DATA_BLOCK "DB2039_TQ"
TITLE = DB2039_TQ
{ S7_Optimized_Access := 'FALSE' }
AUTHOR : HCR
FAMILY : ZeusControl
VERSION : 1.0
//Bloque de datos dispositivo TQ.
   STRUCT
      TQ { S7_SetPoint := 'False'} : Array[0.."N_MAX_DISP_TQ"] of "UDT_ZC_DISP_TQ";
      Mux { S7_SetPoint := 'False'} : Array[0.."N_MAX_MUX_DISP"] of "UDT_ZC_DISP_MUX_TQ";
      Agrup : Array[0.."N_MAX_DISP_AGRUP"] of "UDT_ZC_DISP_AGRUP";
   END_STRUCT;


BEGIN
   TQ[0].Hmi_Estado := 0;
   TQ[0].Estado_TanqueVacio := FALSE;
   TQ[0].Estado_PocisionAltura := FALSE;
   TQ[0].Estado_NivelBajo := FALSE;
   TQ[0].Estado_NivelAlto := FALSE;
   TQ[0].Estado_BocaHombre := FALSE;
   TQ[0].Estado_Mezcla := FALSE;
   TQ[0].Estado_ComOk := FALSE;
   TQ[0].Alarmas_NivelBajo := FALSE;
   TQ[0].Alarmas_NivelAlto := FALSE;
   TQ[0].Alarmas_BocaHombre := FALSE;
   TQ[0].Alarmas_Instrumentacion := FALSE;
   TQ[0].Alarmas_Parametros := FALSE;
   TQ[0].Alarmas_General := FALSE;
   TQ[0].Alarmas_Capacidad := FALSE;
   TQ[0].Orden_Temperatura := FALSE;
   TQ[0].Orden_Agitacion := FALSE;
   TQ[0].Orden_CIP := FALSE;
   TQ[0].Orden_Producto := FALSE;
   TQ[0].Orden_CambioEstado := FALSE;
   TQ[0].Orden_CambioProd1 := FALSE;
   TQ[0].Orden_CambioProd2 := FALSE;
   TQ[0].Config_Habilitar := FALSE;
   TQ[0].Config_HabilitarControlAgitacion := TRUE;
   TQ[0].Config_HabilitarControlTemp := TRUE;
   TQ[0].Config_HabilitarCamisa := TRUE;
   TQ[0].Config_HabilitarAgitador := TRUE;
   TQ[0].Config_HabilitarAlarmas := FALSE;
   TQ[0].Config_HabilitarCalculoVol := FALSE;
   TQ[0].Config_TipoControlTemperatura := FALSE;
   TQ[0].Aux_VisConsignaTemperatura := FALSE;
   TQ[0].Aux_PulsoAlternarAG := FALSE;
   TQ[0].Aux_MemOrdenAgitador := FALSE;
   TQ[0].Aux_MemOrdenTemperatura := FALSE;
   TQ[0].Aux_MemOrdenProducto := FALSE;
   TQ[0].Aux_MemEstadoCIP := FALSE;
   TQ[0].Aux_CipOK := FALSE;
   TQ[0].Orden_ParoControlAgitador := FALSE;
   TQ[0].Orden_ParoControlTemp := FALSE;
   TQ[0].R_Bool_6 := FALSE;
   TQ[0].R_Bool_8 := FALSE;
   TQ[0].Config_GrupoAlarma := 0;
   TQ[0].Estado_EA_Nivel := 0;
   TQ[0].Estado_EA_Temperatura := 0;
   TQ[0].Estado_Tanque := 0;
   TQ[0].Estado_TanqueNuevo := 0;
   TQ[0].Estado_Producto1 := 0;
   TQ[0].Estado_Producto2 := 0;
   TQ[0].Estado_ProductoNuevo := 0;
   TQ[0].Estado_Volumen := 0.0;
   TQ[0].Estado_Presion := 0.0;
   TQ[0].Estado_Altura := 0.0;
   TQ[0].Orden_TipoProducto := 0;
   TQ[0].Orden_ConsignaAgitador := 0.0;
   TQ[0].Config_NumeroEANivel := 0;
   TQ[0].Config_NumeroEATemp := 0;
   TQ[0].Config_NumeroLL := 0;
   TQ[0].Config_NumeroHL := 0;
   TQ[0].Config_NumeroBH := 0;
   TQ[0].Config_NumeroVA := 0;
   TQ[0].Config_NumeroAG := 0;
   TQ[0].Config_TipoAgitacionTiempo := 0;
   TQ[0].Config_TipoAgitacionVelocidad := 0;
   TQ[0].Config_TipoAgitador := 0;
   TQ[0].Config_EscaladoMinTarjeta := 0;
   TQ[0].Config_EscaladoMaxTarjeta := 27648;
   TQ[0].Config_EscaladoMinIngenieria := 0.0;
   TQ[0].Config_EscaladoMaxIngenieria := 0.1;
   TQ[0].Config_ConsignaTemperatura := 0.0;
   TQ[0].Config_HisteresisTemperatura := 0.0;
   TQ[0].Config_VolumenMinControlTemp := 0.0;
   TQ[0].Config_VolumenMaxControlTemp := 0.0;
   TQ[0].Config_VolumenMinControlAgitador := 0.0;
   TQ[0].Config_VolumenMaxControlAgitador := 0.0;
   TQ[0].Config_VolumenTanqueVacio := 0.0;
   TQ[0].Config_VelocidadMinAgitador := 0.0;
   TQ[0].Config_VelocidadMaxAgitador := 0.0;
   TQ[0].Config_VelocidadFijaAgitador := 0.0;
   TQ[0].Config_CapacidadTanque := 0.0;
   TQ[0].Config_DiametroCilindro := 0.0;
   TQ[0].Config_AlturaCilindro := 0.0;
   TQ[0].Config_DiametroConoInferior := 0.0;
   TQ[0].Config_AnguloCono := 0.0;
   TQ[0].Config_AlturaCono := 0.0;
   TQ[0].Tiempos_AgitadorONConsigna := 0;
   TQ[0].Tiempos_AgitadorONActual := 0;
   TQ[0].Tiempos_AgitadorOFFConsigna := 0;
   TQ[0].Tiempos_AgitadorOFFActual := 0;
   TQ[0].Tiempos_TiempoProducto.Hora := 0;
   TQ[0].Tiempos_TiempoProducto.Minuto := 0;
   TQ[0].Tiempos_TiempoProducto.Segundo := 0;
   TQ[0].Tiempos_TiempoLimpio.Hora := 0;
   TQ[0].Tiempos_TiempoLimpio.Minuto := 0;
   TQ[0].Tiempos_TiempoLimpio.Segundo := 0;
   TQ[0].Tiempos_RetTanqueVacio.SP := 5;
   TQ[0].Tiempos_RetTanqueVacio.ET := 0;
   TQ[0].Tiempos_RetTanqueVacio.IN := FALSE;
   TQ[0].Tiempos_RetTanqueVacio.Q := FALSE;
   TQ[0].Aux_ValorTarjetaNivel := 0;
   TQ[0].Aux_ValorIngeneriaTemperatura := 0.0;
   TQ[1].Hmi_Estado := 0;
   TQ[1].Estado_TanqueVacio := TRUE;
   TQ[1].Estado_PocisionAltura := FALSE;
   TQ[1].Estado_NivelBajo := FALSE;
   TQ[1].Estado_NivelAlto := FALSE;
   TQ[1].Estado_BocaHombre := TRUE;
   TQ[1].Estado_Mezcla := FALSE;
   TQ[1].Estado_ComOk := TRUE;
   TQ[1].Alarmas_NivelBajo := FALSE;
   TQ[1].Alarmas_NivelAlto := FALSE;
   TQ[1].Alarmas_BocaHombre := FALSE;
   TQ[1].Alarmas_Instrumentacion := FALSE;
   TQ[1].Alarmas_Parametros := FALSE;
   TQ[1].Alarmas_General := FALSE;
   TQ[1].Alarmas_Capacidad := FALSE;
   TQ[1].Orden_Temperatura := FALSE;
   TQ[1].Orden_Agitacion := FALSE;
   TQ[1].Orden_CIP := FALSE;
   TQ[1].Orden_Producto := FALSE;
   TQ[1].Orden_CambioEstado := FALSE;
   TQ[1].Orden_CambioProd1 := FALSE;
   TQ[1].Orden_CambioProd2 := FALSE;
   TQ[1].Config_Habilitar := TRUE;
   TQ[1].Config_HabilitarControlAgitacion := TRUE;
   TQ[1].Config_HabilitarControlTemp := TRUE;
   TQ[1].Config_HabilitarCamisa := TRUE;
   TQ[1].Config_HabilitarAgitador := TRUE;
   TQ[1].Config_HabilitarAlarmas := FALSE;
   TQ[1].Config_HabilitarCalculoVol := FALSE;
   TQ[1].Config_TipoControlTemperatura := TRUE;
   TQ[1].Aux_VisConsignaTemperatura := FALSE;
   TQ[1].Aux_PulsoAlternarAG := TRUE;
   TQ[1].Aux_MemOrdenAgitador := FALSE;
   TQ[1].Aux_MemOrdenTemperatura := FALSE;
   TQ[1].Aux_MemOrdenProducto := FALSE;
   TQ[1].Aux_MemEstadoCIP := FALSE;
   TQ[1].Aux_CipOK := FALSE;
   TQ[1].Orden_ParoControlAgitador := FALSE;
   TQ[1].Orden_ParoControlTemp := FALSE;
   TQ[1].R_Bool_6 := FALSE;
   TQ[1].R_Bool_8 := FALSE;
   TQ[1].Config_GrupoAlarma := 0;
   TQ[1].Estado_EA_Nivel := 1;
   TQ[1].Estado_EA_Temperatura := 1;
   TQ[1].Estado_Tanque := 2;
   TQ[1].Estado_TanqueNuevo := 1;
   TQ[1].Estado_Producto1 := 0;
   TQ[1].Estado_Producto2 := 0;
   TQ[1].Estado_ProductoNuevo := 1;
   TQ[1].Estado_Volumen := 0.0;
   TQ[1].Estado_Presion := 0.0;
   TQ[1].Estado_Altura := 0.0;
   TQ[1].Orden_TipoProducto := 1;
   TQ[1].Orden_ConsignaAgitador := 0.0;
   TQ[1].Config_NumeroEANivel := 9;
   TQ[1].Config_NumeroEATemp := 4;
   TQ[1].Config_NumeroLL := 0;
   TQ[1].Config_NumeroHL := 0;
   TQ[1].Config_NumeroBH := 8;
   TQ[1].Config_NumeroVA := 33;
   TQ[1].Config_NumeroAG := 4;
   TQ[1].Config_TipoAgitacionTiempo := 1;
   TQ[1].Config_TipoAgitacionVelocidad := 0;
   TQ[1].Config_TipoAgitador := 1;
   TQ[1].Config_EscaladoMinTarjeta := 0;
   TQ[1].Config_EscaladoMaxTarjeta := 27648;
   TQ[1].Config_EscaladoMinIngenieria := 0.0;
   TQ[1].Config_EscaladoMaxIngenieria := 0.1;
   TQ[1].Config_ConsignaTemperatura := 4.0;
   TQ[1].Config_HisteresisTemperatura := 1.0;
   TQ[1].Config_VolumenMinControlTemp := 200.0;
   TQ[1].Config_VolumenMaxControlTemp := 35000.0;
   TQ[1].Config_VolumenMinControlAgitador := 1600.0;
   TQ[1].Config_VolumenMaxControlAgitador := 30000.0;
   TQ[1].Config_VolumenTanqueVacio := 20.0;
   TQ[1].Config_VelocidadMinAgitador := 30.0;
   TQ[1].Config_VelocidadMaxAgitador := 85.0;
   TQ[1].Config_VelocidadFijaAgitador := 35.0;
   TQ[1].Config_CapacidadTanque := 30000.0;
   TQ[1].Config_DiametroCilindro := 0.0;
   TQ[1].Config_AlturaCilindro := 0.0;
   TQ[1].Config_DiametroConoInferior := 0.0;
   TQ[1].Config_AnguloCono := 0.0;
   TQ[1].Config_AlturaCono := 0.0;
   TQ[1].Tiempos_AgitadorONConsigna := 300;
   TQ[1].Tiempos_AgitadorONActual := 0;
   TQ[1].Tiempos_AgitadorOFFConsigna := 1200;
   TQ[1].Tiempos_AgitadorOFFActual := 0;
   TQ[1].Tiempos_TiempoProducto.Hora := 0;
   TQ[1].Tiempos_TiempoProducto.Minuto := 0;
   TQ[1].Tiempos_TiempoProducto.Segundo := 0;
   TQ[1].Tiempos_TiempoLimpio.Hora := 27;
   TQ[1].Tiempos_TiempoLimpio.Minuto := 30;
   TQ[1].Tiempos_TiempoLimpio.Segundo := 25;
   TQ[1].Tiempos_RetTanqueVacio.SP := 25;
   TQ[1].Tiempos_RetTanqueVacio.ET := 25;
   TQ[1].Tiempos_RetTanqueVacio.IN := TRUE;
   TQ[1].Tiempos_RetTanqueVacio.Q := TRUE;
   TQ[1].Aux_ValorTarjetaNivel := 0;
   TQ[1].Aux_ValorIngeneriaTemperatura := 26.19213;
   Mux[0].Habilitar := TRUE;
   Mux[0].ExisteCambio := FALSE;
   Mux[0].MaxVisible := FALSE;
   Mux[0].Index := 0;
   Mux[0].oldIndex := 0;
   Mux[0].TQ.Hmi_Estado := 0;
   Mux[0].TQ.Estado_TanqueVacio := FALSE;
   Mux[0].TQ.Estado_PocisionAltura := FALSE;
   Mux[0].TQ.Estado_NivelBajo := FALSE;
   Mux[0].TQ.Estado_NivelAlto := FALSE;
   Mux[0].TQ.Estado_BocaHombre := FALSE;
   Mux[0].TQ.Estado_Mezcla := FALSE;
   Mux[0].TQ.Estado_ComOk := FALSE;
   Mux[0].TQ.Alarmas_NivelBajo := FALSE;
   Mux[0].TQ.Alarmas_NivelAlto := FALSE;
   Mux[0].TQ.Alarmas_BocaHombre := FALSE;
   Mux[0].TQ.Alarmas_Instrumentacion := FALSE;
   Mux[0].TQ.Alarmas_Parametros := FALSE;
   Mux[0].TQ.Alarmas_General := FALSE;
   Mux[0].TQ.Alarmas_Capacidad := FALSE;
   Mux[0].TQ.Orden_Temperatura := FALSE;
   Mux[0].TQ.Orden_Agitacion := FALSE;
   Mux[0].TQ.Orden_CIP := FALSE;
   Mux[0].TQ.Orden_Producto := FALSE;
   Mux[0].TQ.Orden_CambioEstado := FALSE;
   Mux[0].TQ.Orden_CambioProd1 := FALSE;
   Mux[0].TQ.Orden_CambioProd2 := FALSE;
   Mux[0].TQ.Config_Habilitar := FALSE;
   Mux[0].TQ.Config_HabilitarControlAgitacion := TRUE;
   Mux[0].TQ.Config_HabilitarControlTemp := TRUE;
   Mux[0].TQ.Config_HabilitarCamisa := TRUE;
   Mux[0].TQ.Config_HabilitarAgitador := TRUE;
   Mux[0].TQ.Config_HabilitarAlarmas := FALSE;
   Mux[0].TQ.Config_HabilitarCalculoVol := FALSE;
   Mux[0].TQ.Config_TipoControlTemperatura := FALSE;
   Mux[0].TQ.Aux_VisConsignaTemperatura := FALSE;
   Mux[0].TQ.Aux_PulsoAlternarAG := FALSE;
   Mux[0].TQ.Aux_MemOrdenAgitador := FALSE;
   Mux[0].TQ.Aux_MemOrdenTemperatura := FALSE;
   Mux[0].TQ.Aux_MemOrdenProducto := FALSE;
   Mux[0].TQ.Aux_MemEstadoCIP := FALSE;
   Mux[0].TQ.Aux_CipOK := FALSE;
   Mux[0].TQ.Orden_ParoControlAgitador := FALSE;
   Mux[0].TQ.Orden_ParoControlTemp := FALSE;
   Mux[0].TQ.R_Bool_6 := FALSE;
   Mux[0].TQ.R_Bool_8 := FALSE;
   Mux[0].TQ.Config_GrupoAlarma := 0;
   Mux[0].TQ.Estado_EA_Nivel := 0;
   Mux[0].TQ.Estado_EA_Temperatura := 0;
   Mux[0].TQ.Estado_Tanque := 0;
   Mux[0].TQ.Estado_TanqueNuevo := 0;
   Mux[0].TQ.Estado_Producto1 := 0;
   Mux[0].TQ.Estado_Producto2 := 0;
   Mux[0].TQ.Estado_ProductoNuevo := 0;
   Mux[0].TQ.Estado_Volumen := 0.0;
   Mux[0].TQ.Estado_Presion := 0.0;
   Mux[0].TQ.Estado_Altura := 0.0;
   Mux[0].TQ.Orden_TipoProducto := 0;
   Mux[0].TQ.Orden_ConsignaAgitador := 0.0;
   Mux[0].TQ.Config_NumeroEANivel := 0;
   Mux[0].TQ.Config_NumeroEATemp := 0;
   Mux[0].TQ.Config_NumeroLL := 0;
   Mux[0].TQ.Config_NumeroHL := 0;
   Mux[0].TQ.Config_NumeroBH := 0;
   Mux[0].TQ.Config_NumeroVA := 0;
   Mux[0].TQ.Config_NumeroAG := 0;
   Mux[0].TQ.Config_TipoAgitacionTiempo := 0;
   Mux[0].TQ.Config_TipoAgitacionVelocidad := 0;
   Mux[0].TQ.Config_TipoAgitador := 0;
   Mux[0].TQ.Config_EscaladoMinTarjeta := 0;
   Mux[0].TQ.Config_EscaladoMaxTarjeta := 27648;
   Mux[0].TQ.Config_EscaladoMinIngenieria := 0.0;
   Mux[0].TQ.Config_EscaladoMaxIngenieria := 0.1;
   Mux[0].TQ.Config_ConsignaTemperatura := 0.0;
   Mux[0].TQ.Config_HisteresisTemperatura := 0.0;
   Mux[0].TQ.Config_VolumenMinControlTemp := 0.0;
   Mux[0].TQ.Config_VolumenMaxControlTemp := 0.0;
   Mux[0].TQ.Config_VolumenMinControlAgitador := 0.0;
   Mux[0].TQ.Config_VolumenMaxControlAgitador := 0.0;
   Mux[0].TQ.Config_VolumenTanqueVacio := 0.0;
   Mux[0].TQ.Config_VelocidadMinAgitador := 0.0;
   Mux[0].TQ.Config_VelocidadMaxAgitador := 0.0;
   Mux[0].TQ.Config_VelocidadFijaAgitador := 0.0;
   Mux[0].TQ.Config_CapacidadTanque := 0.0;
   Mux[0].TQ.Config_DiametroCilindro := 0.0;
   Mux[0].TQ.Config_AlturaCilindro := 0.0;
   Mux[0].TQ.Config_DiametroConoInferior := 0.0;
   Mux[0].TQ.Config_AnguloCono := 0.0;
   Mux[0].TQ.Config_AlturaCono := 0.0;
   Mux[0].TQ.Tiempos_AgitadorONConsigna := 0;
   Mux[0].TQ.Tiempos_AgitadorONActual := 0;
   Mux[0].TQ.Tiempos_AgitadorOFFConsigna := 0;
   Mux[0].TQ.Tiempos_AgitadorOFFActual := 0;
   Mux[0].TQ.Tiempos_TiempoProducto.Hora := 0;
   Mux[0].TQ.Tiempos_TiempoProducto.Minuto := 0;
   Mux[0].TQ.Tiempos_TiempoProducto.Segundo := 0;
   Mux[0].TQ.Tiempos_TiempoLimpio.Hora := 0;
   Mux[0].TQ.Tiempos_TiempoLimpio.Minuto := 0;
   Mux[0].TQ.Tiempos_TiempoLimpio.Segundo := 0;
   Mux[0].TQ.Tiempos_RetTanqueVacio.SP := 5;
   Mux[0].TQ.Tiempos_RetTanqueVacio.ET := 0;
   Mux[0].TQ.Tiempos_RetTanqueVacio.IN := FALSE;
   Mux[0].TQ.Tiempos_RetTanqueVacio.Q := FALSE;
   Mux[0].TQ.Aux_ValorTarjetaNivel := 0;
   Mux[0].TQ.Aux_ValorIngeneriaTemperatura := 0.0;
   Mux[1].Habilitar := TRUE;
   Mux[1].ExisteCambio := FALSE;
   Mux[1].MaxVisible := FALSE;
   Mux[1].Index := 0;
   Mux[1].oldIndex := 0;
   Mux[1].TQ.Hmi_Estado := 0;
   Mux[1].TQ.Estado_TanqueVacio := FALSE;
   Mux[1].TQ.Estado_PocisionAltura := FALSE;
   Mux[1].TQ.Estado_NivelBajo := FALSE;
   Mux[1].TQ.Estado_NivelAlto := FALSE;
   Mux[1].TQ.Estado_BocaHombre := FALSE;
   Mux[1].TQ.Estado_Mezcla := FALSE;
   Mux[1].TQ.Estado_ComOk := FALSE;
   Mux[1].TQ.Alarmas_NivelBajo := FALSE;
   Mux[1].TQ.Alarmas_NivelAlto := FALSE;
   Mux[1].TQ.Alarmas_BocaHombre := FALSE;
   Mux[1].TQ.Alarmas_Instrumentacion := FALSE;
   Mux[1].TQ.Alarmas_Parametros := FALSE;
   Mux[1].TQ.Alarmas_General := FALSE;
   Mux[1].TQ.Alarmas_Capacidad := FALSE;
   Mux[1].TQ.Orden_Temperatura := FALSE;
   Mux[1].TQ.Orden_Agitacion := FALSE;
   Mux[1].TQ.Orden_CIP := FALSE;
   Mux[1].TQ.Orden_Producto := FALSE;
   Mux[1].TQ.Orden_CambioEstado := FALSE;
   Mux[1].TQ.Orden_CambioProd1 := FALSE;
   Mux[1].TQ.Orden_CambioProd2 := FALSE;
   Mux[1].TQ.Config_Habilitar := FALSE;
   Mux[1].TQ.Config_HabilitarControlAgitacion := TRUE;
   Mux[1].TQ.Config_HabilitarControlTemp := TRUE;
   Mux[1].TQ.Config_HabilitarCamisa := TRUE;
   Mux[1].TQ.Config_HabilitarAgitador := TRUE;
   Mux[1].TQ.Config_HabilitarAlarmas := FALSE;
   Mux[1].TQ.Config_HabilitarCalculoVol := FALSE;
   Mux[1].TQ.Config_TipoControlTemperatura := FALSE;
   Mux[1].TQ.Aux_VisConsignaTemperatura := FALSE;
   Mux[1].TQ.Aux_PulsoAlternarAG := FALSE;
   Mux[1].TQ.Aux_MemOrdenAgitador := FALSE;
   Mux[1].TQ.Aux_MemOrdenTemperatura := FALSE;
   Mux[1].TQ.Aux_MemOrdenProducto := FALSE;
   Mux[1].TQ.Aux_MemEstadoCIP := FALSE;
   Mux[1].TQ.Aux_CipOK := FALSE;
   Mux[1].TQ.Orden_ParoControlAgitador := FALSE;
   Mux[1].TQ.Orden_ParoControlTemp := FALSE;
   Mux[1].TQ.R_Bool_6 := FALSE;
   Mux[1].TQ.R_Bool_8 := FALSE;
   Mux[1].TQ.Config_GrupoAlarma := 0;
   Mux[1].TQ.Estado_EA_Nivel := 0;
   Mux[1].TQ.Estado_EA_Temperatura := 0;
   Mux[1].TQ.Estado_Tanque := 0;
   Mux[1].TQ.Estado_TanqueNuevo := 0;
   Mux[1].TQ.Estado_Producto1 := 0;
   Mux[1].TQ.Estado_Producto2 := 0;
   Mux[1].TQ.Estado_ProductoNuevo := 0;
   Mux[1].TQ.Estado_Volumen := 0.0;
   Mux[1].TQ.Estado_Presion := 0.0;
   Mux[1].TQ.Estado_Altura := 0.0;
   Mux[1].TQ.Orden_TipoProducto := 0;
   Mux[1].TQ.Orden_ConsignaAgitador := 0.0;
   Mux[1].TQ.Config_NumeroEANivel := 0;
   Mux[1].TQ.Config_NumeroEATemp := 0;
   Mux[1].TQ.Config_NumeroLL := 0;
   Mux[1].TQ.Config_NumeroHL := 0;
   Mux[1].TQ.Config_NumeroBH := 0;
   Mux[1].TQ.Config_NumeroVA := 0;
   Mux[1].TQ.Config_NumeroAG := 0;
   Mux[1].TQ.Config_TipoAgitacionTiempo := 0;
   Mux[1].TQ.Config_TipoAgitacionVelocidad := 0;
   Mux[1].TQ.Config_TipoAgitador := 0;
   Mux[1].TQ.Config_EscaladoMinTarjeta := 0;
   Mux[1].TQ.Config_EscaladoMaxTarjeta := 27648;
   Mux[1].TQ.Config_EscaladoMinIngenieria := 0.0;
   Mux[1].TQ.Config_EscaladoMaxIngenieria := 0.1;
   Mux[1].TQ.Config_ConsignaTemperatura := 0.0;
   Mux[1].TQ.Config_HisteresisTemperatura := 0.0;
   Mux[1].TQ.Config_VolumenMinControlTemp := 0.0;
   Mux[1].TQ.Config_VolumenMaxControlTemp := 0.0;
   Mux[1].TQ.Config_VolumenMinControlAgitador := 0.0;
   Mux[1].TQ.Config_VolumenMaxControlAgitador := 0.0;
   Mux[1].TQ.Config_VolumenTanqueVacio := 0.0;
   Mux[1].TQ.Config_VelocidadMinAgitador := 0.0;
   Mux[1].TQ.Config_VelocidadMaxAgitador := 0.0;
   Mux[1].TQ.Config_VelocidadFijaAgitador := 0.0;
   Mux[1].TQ.Config_CapacidadTanque := 0.0;
   Mux[1].TQ.Config_DiametroCilindro := 0.0;
   Mux[1].TQ.Config_AlturaCilindro := 0.0;
   Mux[1].TQ.Config_DiametroConoInferior := 0.0;
   Mux[1].TQ.Config_AnguloCono := 0.0;
   Mux[1].TQ.Config_AlturaCono := 0.0;
   Mux[1].TQ.Tiempos_AgitadorONConsigna := 0;
   Mux[1].TQ.Tiempos_AgitadorONActual := 0;
   Mux[1].TQ.Tiempos_AgitadorOFFConsigna := 0;
   Mux[1].TQ.Tiempos_AgitadorOFFActual := 0;
   Mux[1].TQ.Tiempos_TiempoProducto.Hora := 0;
   Mux[1].TQ.Tiempos_TiempoProducto.Minuto := 0;
   Mux[1].TQ.Tiempos_TiempoProducto.Segundo := 0;
   Mux[1].TQ.Tiempos_TiempoLimpio.Hora := 0;
   Mux[1].TQ.Tiempos_TiempoLimpio.Minuto := 0;
   Mux[1].TQ.Tiempos_TiempoLimpio.Segundo := 0;
   Mux[1].TQ.Tiempos_RetTanqueVacio.SP := 5;
   Mux[1].TQ.Tiempos_RetTanqueVacio.ET := 0;
   Mux[1].TQ.Tiempos_RetTanqueVacio.IN := FALSE;
   Mux[1].TQ.Tiempos_RetTanqueVacio.Q := FALSE;
   Mux[1].TQ.Aux_ValorTarjetaNivel := 0;
   Mux[1].TQ.Aux_ValorIngeneriaTemperatura := 0.0;
   Agrup[0].AlgunaEnManual := FALSE;
   Agrup[0].AlgunaAlarma := FALSE;
   Agrup[0].NuevaAlarma := FALSE;
   Agrup[1].AlgunaEnManual := FALSE;
   Agrup[1].AlgunaAlarma := FALSE;
   Agrup[1].NuevaAlarma := FALSE;

END_DATA_BLOCK

